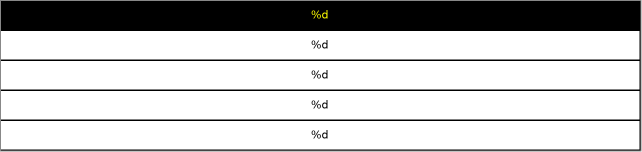
VISUALIZATION CARTON_PICKUP_SHIFT_ELEMENT  // 642x152
VAR_INPUT
	index:		UDINT;
END_VAR
    Rectangle (0,0 640x30), "%d", text variable: wu_cartonPickup_shiftRegister_debug.shift_debug[index].step_id
    Rectangle (0,30 640x30), "%d", text variable: wu_cartonPickup_shiftRegister_debug.shift_debug[index].status.0, colour toggle: wu_cartonPickup_shiftRegister_debug.shift_debug[index].status.0
    Rectangle (0,60 640x30), "%d", text variable: wu_cartonPickup_shiftRegister_debug.shift_debug[index].reject_reason
    Rectangle (0,90 640x30), "%d", text variable: wu_cartonPickup_shiftRegister_debug.shift_debug[index].status.4, colour toggle: wu_cartonPickup_shiftRegister_debug.shift_debug[index].status.4
    Rectangle (0,120 640x30), "%d", text variable: wu_cartonPickup_shiftRegister_debug.shift_debug[index].equipment_number
END_VISUALIZATION

(* stored: Version 1.1.0.1, ProductVersion 3.1.4024.3
   Visu CARTON_PICKUP_SHIFT_ELEMENT: Id {16a51b4a-a10e-416c-b2e6-a81f2298c9cc} *)
